// TIA Portal V21 export
VAR_GLOBAL   // PLC tag table "OutputDigitali"
   ZonaSterilizzatore_AllarmeAcustico AT %Q0.0 : Bool;
   ZonaSterilizzatore_AllarmeVisivo AT %Q0.1 : Bool;
   ZonaSterilizzatore_SegnalazioneSterilizzazione AT %Q0.2 : Bool;
   ZonaSterilizzatore_SegnalazioneProduzione AT %Q0.3 : Bool;
   ZonaSterilizzatore_SegnalazioneLavaggio AT %Q0.4 : Bool;
   ZonaSterilizzatore_SpiaMarcia AT %Q0.5 : Bool;
   ZonaSterilizzatore_SpiaRecupero AT %Q0.6 : Bool;
   ZonaSterilizzatore_SpiaReset AT %Q0.7 : Bool;
   Agitatore_ComandoMarcia AT %Q1.0 : Bool;
   PompaMono_ComandoMarcia AT %Q1.1 : Bool;
   PompaMono_ComandoServoventola AT %Q1.2 : Bool;
   CentrifugaLavaggio_ComandoMarcia AT %Q1.3 : Bool;
   PompaPistoni_ComandoMarcia AT %Q1.4 : Bool;
   PompaPistoni_Servoventola_ComandoMarcia AT %Q1.5 : Bool;
   PompaOlio_ComandoMarcia AT %Q1.6 : Bool;
   PompaRicircoloAcqua_ComandoMarcia AT %Q1.7 : Bool;
   PompaRilancioTorre_ComandoMarcia AT %Q2.0 : Bool;
   PompaPistoni_Aspiratore_Marcia AT %Q2.1 : Bool;
   PompaPistoni_ResetInverter AT %Q2.2 : Bool;
   Valvola_A_ComandoPositivo AT %Q2.3 : Bool;
   Valvola_A1_ComandoPositivo AT %Q2.4 : Bool;
   Valvola_B_ComandoPositivo AT %Q2.5 : Bool;
   Valvola_C_ComandoPositivo AT %Q2.6 : Bool;
   Valvola_D_ComandoPositivo AT %Q2.7 : Bool;
   Valvola_E_ComandoPositivo AT %Q3.0 : Bool;
   Valvola_E1_ComandoPositivo AT %Q3.1 : Bool;
   Valvola_F_ComandoPositivo AT %Q3.2 : Bool;
   Valvola_G_ComandoPositivo AT %Q3.3 : Bool;
   Valvola_H_ComandoPositivo AT %Q3.4 : Bool;
   Valvola_H1_ComandoPositivo AT %Q3.5 : Bool;
   Valvola_Z_ComandoPositivo AT %Q3.6 : Bool;
   "A3.7" AT %Q3.7 : Bool;
   Valvola_Y_ComandoPositivo AT %Q4.0 : Bool;
   Valvola_Y1_ComandoPositivo AT %Q4.1 : Bool;
   Valvola_Y2_ComandoPositivo AT %Q4.2 : Bool;
   Valvola_J_ComandoPositivo AT %Q4.3 : Bool;
   Valvola_X_ComandoPositivo AT %Q4.4 : Bool;
   Valvola_N_ComandoPositivo AT %Q4.5 : Bool;
   Valvola_N1_ComandoPositivo AT %Q4.6 : Bool;
   "Valvola_EV103.6_ComandoPositivo" AT %Q4.7 : Bool;
   Consenso_ACFT_ImpiantoInSterilizzazione AT %Q5.0 : Bool;
   Consenso_ACFT_ImpiantoInLavaggio AT %Q5.1 : Bool;
   Consenso_ACFT_ImpulsiPompaPistoni AT %Q5.2 : Bool;
   Consenso_ACFT_ImpiantoInProduzione AT %Q5.3 : Bool;
   Consenso_ACFT_ProdottoDisponibile AT %Q5.4 : Bool;
   Consenso_AQCI_ChiamataProdotto AT %Q5.5 : Bool;
   "A5.6" AT %Q5.6 : Bool;
   "A5.7" AT %Q5.7 : Bool;
   Valvola_XXX_ComandoPositivo AT %Q6.0 : Bool;
   Valvola_XX_ComandoPositivo AT %Q6.1 : Bool;
   Valvola_L_ComandoPositivo AT %Q6.2 : Bool;
   Valvola_R_ComandoPositivo AT %Q6.3 : Bool;
   Valvola_Z1_ComandoPositivo AT %Q6.4 : Bool;
   Valvola_I_ComandoPositivo AT %Q6.5 : Bool;
   ValvolaIntercetto_RiscaldAcqua_ComandoPositivo AT %Q6.7 : Bool;
   "A7.0" AT %Q7.0 : Bool;
   "A7.1" AT %Q7.1 : Bool;
   "A7.2" AT %Q7.2 : Bool;
   "A7.3" AT %Q7.3 : Bool;
   "A7.4" AT %Q7.4 : Bool;
   "A7.5" AT %Q7.5 : Bool;
   "A7.6" AT %Q7.6 : Bool;
   "A7.7" AT %Q7.7 : Bool;
   Valvola_X2_ComandoPositivo AT %Q6.6 : Bool;
END_VAR
